INTERFACE I_AxisHome EXTENDS I_Base

METHOD Home
VAR_INPUT
END_VAR
END_METHOD

END_INTERFACE

(* stored: Version 1.1.0.1, ProductVersion 3.1.4026.18
   Itf I_AxisHome: Id {049b3ba0-b295-43f0-be24-e10097b70ce7}
   Method Home: Id {94d26bc7-8fa6-4697-9008-21ad5a0d0f62} *)
